FUNCTION_BLOCK PUBLISH_2 (* Two-Variable Publisher *)
  (* Standard: 61499-1; Classification: Communications; Function: 2-variable publisher *)
  (* Version 0.1, 2008-06-04, JHC, Holobloc Inc, Updated DOCTYPE. *)
  (* Version 0.0, 2001-04-14, JHC, Rockwell Automation, First XML version *)
  (* Compiler header: package fb.rt.net; *)
  (* Compiler Java IBM VisualAge 3.0 *)
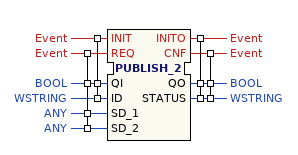
  EVENT_INPUT
    INIT WITH QI, ID; (* Service Initialization *)
    REQ WITH QI, SD_1, SD_2; (* Service Request *)
  END_EVENT
  EVENT_OUTPUT
    INITO WITH QO, STATUS; (* Initialization Confirm *)
    CNF WITH QO, STATUS; (* Service Confirmation *)
  END_EVENT
  VAR_INPUT
    QI : BOOL; (* Event Input Qualifier *)
    ID : WSTRING; (* Connection Identifier *)
    SD_1 : ANY; (* Data to Send *)
    SD_2 : ANY; (* Data to Send *)
  END_VAR
  VAR_OUTPUT
    QO : BOOL; (* Event Output Qualifier *)
    STATUS : WSTRING; (* Service Status *)
  END_VAR
  SERVICE PUBLISH_2/SUBSCRIBE_2 (* Data Publication Service *)
    SEQUENCE normal_establishment
      PUBLISH_2.INIT+(ID) -> PUBLISH_2.INITO+();
      SUBSCRIBE_2.INIT+(ID) -> SUBSCRIBE_2.INITO+();
    END_SEQUENCE
    SEQUENCE publisher_rejected_establishment
      PUBLISH_2.INIT+(ID) -> PUBLISH_2.INITO-(STATUS);
    END_SEQUENCE
    SEQUENCE subscriber_rejected_establishment
      SUBSCRIBE_2.INIT+(ID) -> SUBSCRIBE_2.INITO-(STATUS);
    END_SEQUENCE
    SEQUENCE normal_data_transfer
      PUBLISH_2.REQ+(SD_1,SD_2) -> SUBSCRIBE_2.IND+(RD_1,RD_2);
      -> PUBLISH_2.CNF+();
      SUBSCRIBE_2.RSP+();
    END_SEQUENCE
    SEQUENCE data_transfer_error
      PUBLISH_2.REQ+(SD_1,SD_2) -> SUBSCRIBE_2.IND-(STATUS);
      -> PUBLISH_2.CNF+();
    END_SEQUENCE
    SEQUENCE publisher_initiated_disconnect
      PUBLISH_2.INIT-() -> SUBSCRIBE_2.INITO-(STATUS);
      -> PUBLISH_2.INITO-(STATUS);
    END_SEQUENCE
    SEQUENCE subscriber_initiated_disconnect
      SUBSCRIBE_2.INIT-() -> SUBSCRIBE_2.INITO-(STATUS);
    END_SEQUENCE
    SEQUENCE system_publisher_disconnect
      -> PUBLISH_2.INITO-(STATUS);
      -> SUBSCRIBE_2.INITO-(STATUS);
    END_SEQUENCE
    SEQUENCE system_subscriber_disconnect
      -> SUBSCRIBE_2.INITO-(STATUS);
    END_SEQUENCE
  END_SERVICE
END_FUNCTION_BLOCK
